// TIA Portal V17 export
// export: Created 2024-09-26T08:51:31.9404074Z, ExportSetting WithDefaults, DisplayName Totally Integrated Automation Portal, DisplayVersion V17, DisplayName TIA Portal Openness, DisplayVersion V17, DisplayName TIA Portal Version Control Interface, DisplayVersion V17, DisplayName STEP 7 Professional, DisplayVersion V17, DisplayName STEP 7 Safety, DisplayVersion V17, DisplayName WinCC Advanced / Unified PC, DisplayVersion V17
ORGANIZATION_BLOCK "Main"   // OB1, LAD, ProgramCycle
TITLE = "Main Program Sweep (Cycle)"
{ S7_Optimized_Access := 'TRUE' }
VERSION : 0.1
// stored: AutoNumber true, IsIECCheckEnabled false, SetENOAutomatically false
   VAR_INPUT
      Initial_Call : Bool;   // Initial call of this OB
      Remanence : Bool;   // =True, if remanent data are available
   END_VAR
BEGIN

REGION Network 1
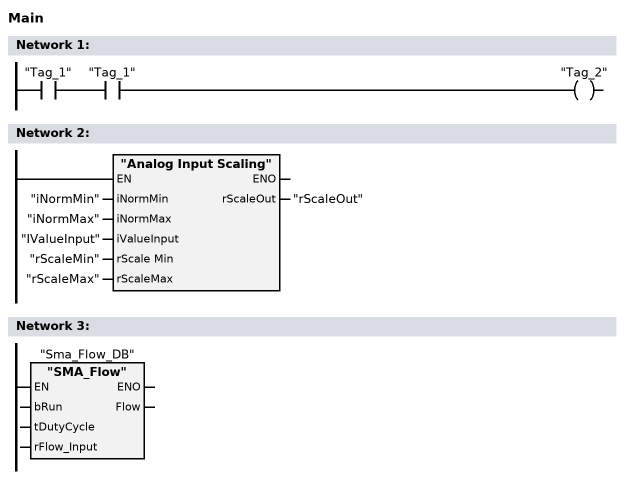
   RUNG wire#powerrail
      Contact( "Tag_1" )
      Contact( "Tag_1" )
      Coil( "Tag_2" )
   END_RUNG
   // the same network as SCL:
   "Tag_2" := "Tag_1" AND "Tag_1";
END_REGION

REGION Network 2
   RUNG wire#powerrail
      "Analog Input Scaling"(iNormMin := "iNormMin", iNormMax := "iNormMax", iValueInput := "IValueInput", "rScale Min" := "rScaleMin", rScaleMax := "rScaleMax", rScaleOut => "rScaleOut")
   END_RUNG
   // the same network as SCL:
   "Analog Input Scaling"(iNormMin := "iNormMin",
                          iNormMax := "iNormMax",
                          iValueInput := "IValueInput",
                          "rScale Min" := "rScaleMin",
                          rScaleMax := "rScaleMax",
                          rScaleOut => "rScaleOut");
END_REGION

REGION Network 3
   RUNG wire#powerrail
      "Sma_Flow_DB"(bRun :=, tDutyCycle :=, rFlow_Input :=, Flow =>)
   END_RUNG
   // the same network as SCL:
   "Sma_Flow_DB"();   // "SMA_Flow"
END_REGION
END_ORGANIZATION_BLOCK
